(* CODESYS project tesina_IOT.project

Project tree, tasks and I/O mapping:
  Device : CODESYS Control Win V3, 3S - Smart Software Solutions GmbH, version 3.5.12.40
    application Application
      libraries: Standard, * (System); VisuDialogs, * (System)
      task MainTask (cyclic, interval t#20ms, priority 1) calls PLC_PRG
      task VISU_TASK (cyclic, interval 100 ms, priority 31) calls VisuElems.Visu_Prg
      program PLC_PRG [SFC]: Main_active
      function block OOM [ST]
      function block SWITCHER [ST]
      function block ARM_GRID [ST]
      function block ARM_CONTROLLER [ST]
      function block MAIN_CONTROLLER [ST]
      visualisation Visualization
      image pool ImagePool
  text list GlobalTextList
  5ce3da45-db07-42e7-a21c-a00fff4ed8f6|C:\Users\marco\Downloads\Telegram Desktop\abbassato con fusto DX.png
  5ce3da45-db07-42e7-a21c-a00fff4ed8f6|C:\Users\marco\Downloads\Telegram Desktop\abbassato con fusto SX.png
  5ce3da45-db07-42e7-a21c-a00fff4ed8f6|C:\Users\marco\Downloads\Telegram Desktop\alzato con fusto giù DX posizione A.png
  5ce3da45-db07-42e7-a21c-a00fff4ed8f6|C:\Users\marco\Downloads\Telegram Desktop\alzato con fusto giù DX posizione B.png
  5ce3da45-db07-42e7-a21c-a00fff4ed8f6|C:\Users\marco\Downloads\Telegram Desktop\alzato con fusto giù DX posizione C.png
  5ce3da45-db07-42e7-a21c-a00fff4ed8f6|C:\Users\marco\Downloads\Telegram Desktop\alzato con fusto giù SX.png
  5ce3da45-db07-42e7-a21c-a00fff4ed8f6|C:\Users\marco\Downloads\Telegram Desktop\alzato con fusto su DX.png
  5ce3da45-db07-42e7-a21c-a00fff4ed8f6|C:\Users\marco\Downloads\Telegram Desktop\alzato con fusto su SX.png
  5ce3da45-db07-42e7-a21c-a00fff4ed8f6|C:\Users\marco\Downloads\Telegram Desktop\alzato no fusto SX.png
  5ce3da45-db07-42e7-a21c-a00fff4ed8f6|C:\Users\marco\Downloads\Telegram Desktop\alzato posizione 0 - Copia.png
  5ce3da45-db07-42e7-a21c-a00fff4ed8f6|C:\Users\marco\Downloads\Telegram Desktop\alzato con fusto su DX A.png
  5ce3da45-db07-42e7-a21c-a00fff4ed8f6|C:\Users\marco\Downloads\Telegram Desktop\alzato con fusto su DX B.png
  5ce3da45-db07-42e7-a21c-a00fff4ed8f6|C:\Users\marco\Downloads\Telegram Desktop\alzato con fusto su DX C.png
  5ce3da45-db07-42e7-a21c-a00fff4ed8f6|C:\Users\marco\Downloads\Telegram Desktop\alzato con fusto giù DX.png
  5ce3da45-db07-42e7-a21c-a00fff4ed8f6|C:\Users\marco\Desktop\alzato con fusto pos 0.png
*)

// Device/Application/PLC_PRG
PROGRAM PLC_PRG
VAR
	end : OOM();
	grid : ARM_GRID();
	//sensors and stuff
	barcode, geiger : SWITCHER();
	weight: OOM(); //sensor
	start_button: OOM(); //button
	reset_button: OOM(); //button
	light: OOM(); //emergency ligh
	c0 : MAIN_CONTROLLER();
	c1 : ARM_CONTROLLER();
END_VAR

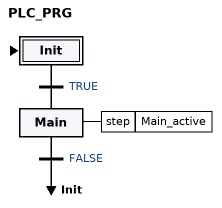
INITIAL_STEP Init:
END_STEP
TRANSITION FROM Init TO Main
    := TRUE;
END_TRANSITION
STEP Main:
    Main_active(N);  // step action
END_STEP
TRANSITION FROM Main TO Init
    := FALSE;
END_TRANSITION

ACTION Main_active:
//INIT
//third level
barcode();
geiger();
weight(); 
start_button();
reset_button();
light();
end();
grid();


c1.grid_input := grid;
c1.hand_input := end;
c1();
end := c1.hand_output;
grid := c1.grid_output;

//first level
c0.arm_controller_input := c1;
c0.barcode_input := barcode;
c0.geiger_input := geiger;
c0.light_input := light;

//solo input per c0
c0.reset_button_input := reset_button;
c0.start_button_input := start_button;
c0.weight_input := weight;

c0();
c1 := c0.arm_controller_output;
barcode := c0.barcode_output;
geiger := c0.geiger_output;
light := c0.light_output;
END_ACTION

END_PROGRAM

// Device/Application/OOM
FUNCTION_BLOCK OOM
// if this class will be used as controller for the  robot hand, we'll assume false as OPEN HAND and true as CLOSED HAND
VAR_INPUT
	stato_in : BOOL := FALSE;
END_VAR
VAR_OUTPUT
	stato_out : BOOL := FALSE;
END_VAR
VAR
	stato : INT := 0;
END_VAR

// 0 idle, 1 off, 2 on
CASE stato OF
	0:
		stato := 1;
		stato_out := FALSE;
		stato_in := FALSE;
	;
	1:
		IF stato_in THEN
			stato := 2;
			stato_out := TRUE;
		END_IF
	;
	2:
		IF NOT stato_in THEN
			stato := 1;
			stato_out := FALSE;
		END_IF
	;
END_CASE

END_FUNCTION_BLOCK

// Device/Application/ARM_GRID
FUNCTION_BLOCK ARM_GRID
VAR_INPUT
	direction : STRING := ''; // 0 or A or B or C or X
END_VAR
VAR_OUTPUT
	current_basket : STRING := '0';
END_VAR
VAR
	status : INT := 1;
	t:TON();
END_VAR

// 0 idle, 1 off, 2 on
CASE status OF
	0: //TR0
		current_basket := 'tr0';
		t(IN := TRUE, PT := T#10S); // emulating transition
		IF  (t.Q = TRUE) THEN // basket 0 reached
			t(IN := FALSE);
			status := 1; //move to starting point on init
		END_IF
	;
	1: // slot 0 starting point
		current_basket := '0';
		IF direction = 'trX' THEN // waiting for new direction's instructions (can be only X from this point)
			status := 5;
		END_IF
	;
	2: // slot A
		t(IN := TRUE, PT := T#10S); // emulating transition
		current_basket := 'trA';
		IF  (t.Q = TRUE) THEN // basket A reached
			t(IN := FALSE);
			status := 7;
		END_IF
	;
	3: // slot B
		t(IN := TRUE, PT := T#10S); // emulating transition
		current_basket := 'trB';
		IF  (t.Q = TRUE) THEN // basket B reached
			t(IN := FALSE);
			status := 8;
		END_IF
	;
	4: // slot C
		t(IN := TRUE, PT := T#10S); // emulating transition
		current_basket := 'trC';
		IF  (t.Q = TRUE) THEN // basket C reached
			t(IN := FALSE);
			status := 9;
		END_IF
	;
	5: // slot X -> grabbing pack
		current_basket := 'trX';
		t(IN := TRUE, PT := T#10S); // emulating transition
		IF  (t.Q = TRUE) THEN // basket X reached
			t(IN := FALSE);
			status := 6;
		END_IF
	;
	6:
		current_basket := 'X';
		// waiting for new direction's instructions (can be everything from this point)
		IF direction = 'trA' THEN
			status := 2;
		ELSIF  direction = 'trB' THEN
			status := 3;
		ELSIF  direction = 'trC' THEN
			status := 4;
		ELSIF  direction = 'tr0' THEN
			status := 0;
		END_IF
	;
	7: //A reached
	current_basket := 'A';
	IF direction = 'tr0' THEN
		status := 0; // to basket number 0
	END_IF
	;
	8: //B reached
	current_basket := 'B';
	IF direction = 'tr0' THEN
		status := 0; // to basket number 0
	END_IF
	;
	9: //C reached
	IF direction = 'tr0' THEN
		status := 0; // to basket number 0
	END_IF
	;
END_CASE

END_FUNCTION_BLOCK

// Device/Application/SWITCHER
FUNCTION_BLOCK SWITCHER
VAR_INPUT
	//active : BOOL := FALSE; //on -> scanning, off -> turned off
	type_simulation : STRING := '';
END_VAR
VAR_OUTPUT
	basket : STRING := 'U'; //values: U (undefined), A, B, C
END_VAR
VAR
	t:TON();
END_VAR

// 0 idle, 1 off, 2 on

IF type_simulation <> 'A' AND type_simulation <> 'B' AND type_simulation <> 'C' THEN
	basket := 'U';
ELSE
	basket := type_simulation;
END_IF

END_FUNCTION_BLOCK

// Device/Application/MAIN_CONTROLLER
FUNCTION_BLOCK MAIN_CONTROLLER
VAR_INPUT
	arm_controller_input : ARM_CONTROLLER();
	barcode_input, geiger_input : SWITCHER();
	weight_input: OOM(); //sensor
	
	start_button_input: OOM(); //button
	reset_button_input: OOM(); //button
	light_input: OOM(); //emergency light
END_VAR
VAR_OUTPUT
	arm_controller_output : ARM_CONTROLLER();
	barcode_output, geiger_output : SWITCHER();

	light_output: OOM(); //emergency light
END_VAR
VAR
	console : STRING := 'init';
	barcode_res, gaiger_res : STRING;
	A_counter, B_counter, C_counter : INT;
	status : INT := 0;
	t:TON();
	//var for UI. true -> invisible
	UI_x, UI_x_grab, UI_x_hold, UI_0, UI_0_W, UI_a_hold, UI_b_hold, UI_c_hold, UI_abc_landed, UI_abc_drop : BOOL := TRUE;
END_VAR

CASE status OF
	0: // INIT
		UI_0 := FALSE;
		IF weight_input.stato_out THEN
			status := 1;
			console := 'sensore di peso attivato, aspettando operatore';
		ELSIF start_button_input.stato_out THEN
			status := 8; //ERROR!
			console := 'bottone premuto ma nulla sul basket. errore!';
		END_IF
		//UI
		IF status <> 0 THEN 
			UI_0 := TRUE;
		END_IF
	;
	1: //s0, weight sensor
		UI_0_W := FALSE;
		IF start_button_input.stato_out THEN
			console := 'bottone premuto, spostamento braccio verso X';
			arm_controller_input.direction := 'trX';
			status := 2;
		END_IF
		//UI
		IF status <> 1 THEN 
			UI_0_W := TRUE;
		END_IF
	;
	2: //TRX
		UI_x := FALSE;
		IF arm_controller_input.position = 'X' THEN
			console := 'braccio ha raggiunto X';
			status := 3;
		END_IF
		//UI
		IF status <> 2 THEN 
			UI_x := TRUE;
		END_IF
	;
	3: //x, timer for grabbing package
		UI_x_grab := FALSE;
		t(IN := TRUE, PT := T#5S);
		console := 'attesa di 5 secondi per la presa del pacco (gestita da c1).';
		IF  (t.Q = TRUE) THEN
			t(IN := FALSE);
			status := 4;
		END_IF
		//UI
		IF status <> 3 THEN
			UI_x_grab := TRUE;	
		END_IF
	;
	4: //scan
		UI_x_hold := FALSE;
		IF barcode_input.basket = 'A' OR barcode_input.basket = 'B' OR barcode_input.basket = 'C' THEN
			console := 'scansione barcode pacco completata correttamente';
			status := 5;
			barcode_res := barcode_input.basket;
		ELSIF barcode_input.basket = 'U' THEN
			console := 'scansione barcode fallita, pacco uknown';
			status := 9;
		END_IF
		//UI
		IF status <> 4 THEN
			UI_x_hold := TRUE;			
		END_IF
	;
	5: //verify
		UI_x_hold := FALSE;
		gaiger_res := geiger_output.basket;
		IF gaiger_res = 'U' OR gaiger_res <> barcode_res THEN
			console := 'scansione radioattività fallita, unknown o diverso dal barcode';
			status := 9;
		ELSIF gaiger_res = 'A' THEN //package A
			console := 'scansioni completate: analisi pacco A';
			IF A_counter > 4 THEN
				status := 9; // full
				console := 'nastro trasportatore A pieno. errore';
			ELSE
				A_counter := A_counter + 1;
				arm_controller_input.direction := 'trA';
				console := 'avviato braccio verso nastro A, incrementato contatore';
				status := 10; 
			END_IF
		ELSIF gaiger_res = 'B' THEN //package B
			console := 'scansioni completate: analisi pacco B';
			IF B_counter > 4 THEN
				console := 'nastro trasportatore B pieno. errore';
				status := 9; // full
			ELSE
				B_counter := B_counter + 1;
				arm_controller_input.direction := 'trB';
				status := 11; 
				console := 'avviato braccio verso nastro B, incrementato contatore';
			END_IF
		ELSIF gaiger_res = 'C' THEN //package C
			console := 'scansioni completate: analisi pacco C';
			IF C_counter > 4 THEN
				status := 9; // full
				console := 'nastro trasportatore C pieno. errore';
			ELSE
				C_counter := C_counter + 1;
				arm_controller_input.direction := 'trC';
				status := 12; 
				console := 'avviato pacco verso nastro C, incrementato contatore';
			END_IF
		END_IF
		//UI
		IF status <> 5 THEN
			UI_x_hold := TRUE;			
		END_IF
	;
	6:
		UI_abc_landed := FALSE;
		console := 'attesa 5 secondi sgancio pacco in postazione';
		t(IN := TRUE, PT := T#5S);
		IF  (t.Q = TRUE) THEN
			t(IN := FALSE);
			status := 7;
		END_IF
		//UI
		IF status <> 6 THEN 
			UI_abc_landed := TRUE;
		END_IF
	;
	7:
		UI_abc_drop := FALSE;
		console := 'sgancio completato, redirezionamento braccio verso tr0';
		arm_controller_input.direction := 'tr0';
		status := 13;
		//UI
		IF status <> 7 THEN 
			UI_abc_drop := TRUE;
		END_IF
	;
	
	/////////////////
	// ERROR SECTION
	////////////////
	8: //B0 ERR, start_button pushed before weight sensor is ok
		UI_0 := FALSE;
		light_input.stato_in := TRUE;
		IF reset_button_input.stato_out THEN
			light_input.stato_in := FALSE;
			console := 'bottone di reset premuto, siamo tornati ad init';
			status := 0;
		END_IF
		//UI
		IF status <> 8 THEN 
			UI_0 := TRUE;
		END_IF
	;
	9: //ERROR come case 8 ma riporto il braccio in posizione 0 e quando resetto assumo di aver svuotato i rulli
		UI_0 := FALSE;
		light_input.stato_in := TRUE;
		arm_controller_input.direction := 'tr0'; //questo dovrebbe essere colto come errore da arm controller, passaggio da X -> tr0
		IF reset_button_input.stato_out AND arm_controller_input.position = '0' THEN
			light_input.stato_in := FALSE;
			A_counter := 0;
			B_counter := 0;
			C_counter := 0;
			console := 'braccio è in 0, slot svuotati, bottone di reset premuto, siamo tornati ad init';
			status := 0;
		END_IF
		//UI
		IF status <> 9 THEN 
			UI_0 := TRUE;
		END_IF
	;
	//////////////
	// END ERRORS
	/////////////
	
	10:
		UI_a_hold := FALSE;
		IF arm_controller_input.position = 'A' THEN
			console := 'postazione A raggiunta';
			status := 6;
		END_IF
		//UI
		IF status <> 10 THEN
			UI_a_hold := TRUE;			
		END_IF
	;
	11:
		UI_b_hold := FALSE;
		IF arm_controller_input.position = 'B' THEN
			console := 'postazione B raggiunta';
			status := 6;
		END_IF
		//UI
		IF status <> 11 THEN
			UI_b_hold := TRUE;			
		END_IF
	;
	12:
		UI_c_hold := FALSE;
		IF arm_controller_input.position = 'C' THEN
			console := 'postazione C raggiunta';
			status := 6;
		END_IF
		//UI
		IF status <> 12 THEN
			UI_c_hold := TRUE;			
		END_IF
	;
	13:
		UI_0 := FALSE;
		IF arm_controller_input.position = '0' THEN
			console := 'postazione 0 raggiunta. siamo tornati ad init';
			status := 0;
		END_IF
		//UI
		IF status <> 13 THEN
			UI_0 := TRUE;			
		END_IF
	;
END_CASE

//updating values
arm_controller_output := arm_controller_input;
barcode_output := barcode_input;
geiger_output := geiger_input;
light_output := light_input;

END_FUNCTION_BLOCK

// Device/Application/ARM_CONTROLLER
FUNCTION_BLOCK ARM_CONTROLLER
VAR_INPUT
	direction : STRING := 'INIT';
	grid_input : ARM_GRID();
	hand_input : OOM();
	//c0_input : MAIN_CONTROLLER();
END_VAR
VAR_OUTPUT
	position : STRING := '';
	grid_output : ARM_GRID();
	hand_output : OOM();
	//c0_output : MAIN_CONTROLLER();
END_VAR
VAR
	status : INT := 0;
END_VAR

CASE status OF
	0:	//INIT
		IF direction = 'trX' THEN //moving grid to trX and 
			grid_input.direction := 'trX';
			status := 1;
		END_IF
	;
	1: //TRX
		IF grid_input.current_basket = 'X' THEN
			hand_input.stato_in := TRUE;
			position := 'X';
			status := 2;
		END_IF
	;
	2: //X
		IF direction = 'trA' THEN //moving grid to trA 
			grid_input.direction := 'trA';
			status := 3; //A
		ELSIF direction = 'trB' THEN //moving grid to trB  
			grid_input.direction := 'trB';
			status := 4; //B
		ELSIF direction = 'trC' THEN //moving grid to trC  
			grid_input.direction := 'trC';
			status := 5; //C
		ELSIF direction = 'tr0' THEN //ERROR DETECTED!! 
			//it's like case 6
			grid_input.direction := 'tr0';
			status := 7; // waiting for destination reached
		END_IF
	;
	3: //A
		IF grid_input.current_basket = 'A' THEN
			hand_input.stato_in := FALSE; 
			position := 'A';
			status := 6; //GOING TO WAIT RESET
		END_IF
	;
	4: //B
		IF grid_input.current_basket = 'B' THEN
			hand_input.stato_in := FALSE; 
			position := 'B';
			status := 6; //GOING TO WAIT RESET
		END_IF		
	;
	5: //C
		IF grid_input.current_basket = 'C' THEN
			hand_input.stato_in := FALSE; 
			position := 'C';
			status := 6; //GOING TO WAIT RESET
		END_IF
	;
	6: //WAITING FOR RESET
		IF direction = 'tr0' THEN //moving grid to tr0 
			grid_input.direction := 'tr0';
			status := 7; //WAITING FOR TR0
		END_IF
	;
	7: // WHEN 0 IS REACHED WE SWITCH TO INIT
		IF grid_input.current_basket = '0' THEN
			position := '0';
			status := 0; // init
		END_IF
	;	
END_CASE

grid_output := grid_input;
hand_output := hand_input;

END_FUNCTION_BLOCK

// Device/Application/Visualization
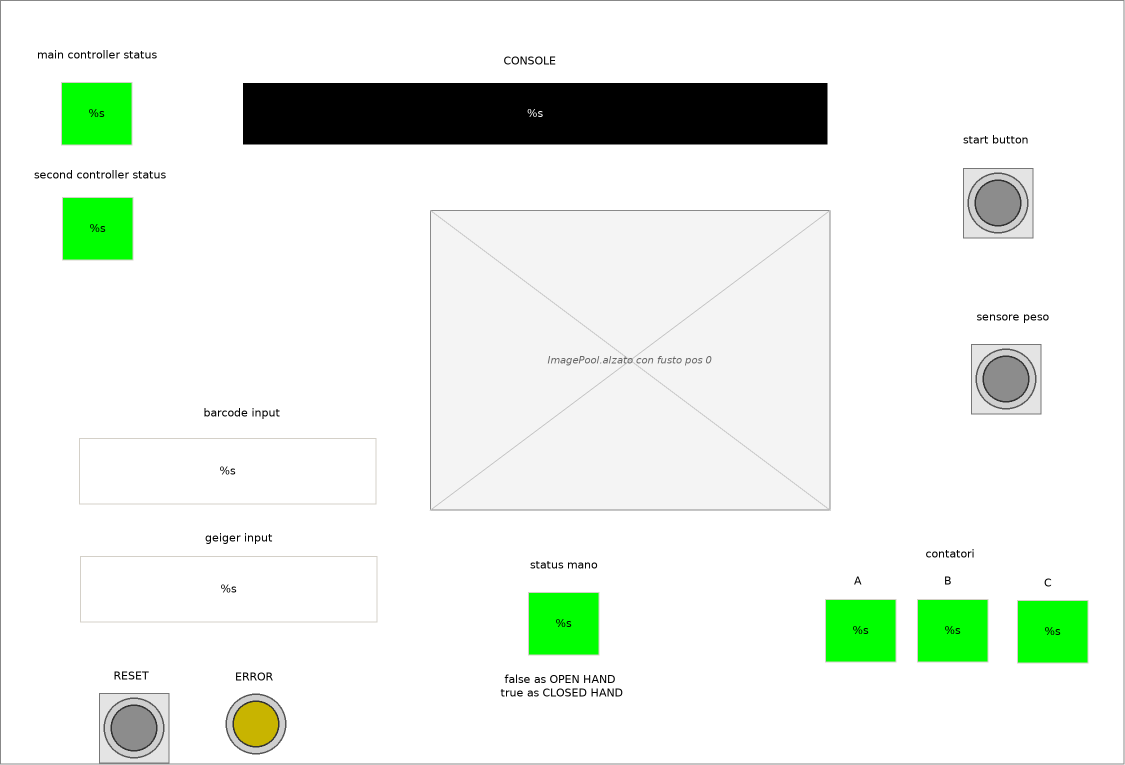
VISUALIZATION Visualization  // 1125x765
    Textfield (61,82 71x63), "%s", text variable: PLC_PRG.c0.status
    Textfield (79,438 297x66), "%s", text variable: PLC_PRG.barcode.type_simulation
        OnMouseClick: write the text variable via Default
    Textfield (80,556 297x66), "%s", text variable: PLC_PRG.geiger.type_simulation
        OnMouseClick: write the text variable via Default
    Label (167,398 150x30), "barcode input"
    Label (164,523 150x30), "geiger input"
    Label (22,40 150x30), "main controller status"
    PushSwitchLed (963,168 70x70), variable: PLC_PRG.start_button.stato_in, behaviour: TOGGLE, style: Switch-PushSwitchLed-Gray
    Label (921,125 150x30), "start button"
    Label (938,302 150x30), "sensore peso"
    PushSwitchLed (971,344 70x70), variable: PLC_PRG.weight.stato_in, behaviour: TOGGLE, style: Switch-PushSwitchLed-Gray
    Textfield (62,197 71x63), "%s", text variable: PLC_PRG.c1.status
    Label (25,160 150x30), "second controller status"
    Textfield (242,82 586x63), "%s", text variable: PLC_PRG.c0.console
    Label (455,46 150x30), "CONSOLE"
    Textfield (528,592 71x63), "%s", text variable: PLC_PRG.end.stato_out
    Label (489,550 150x30), "status mano"
    Textfield (825,599 71x63), "%s", text variable: PLC_PRG.c0.A_counter
    Label (783,566 150x30), "A"
    PushSwitchLed (99,693 70x70), variable: PLC_PRG.reset_button.stato_in, behaviour: TOGGLE, style: Switch-PushSwitchLed-Gray
    Label (56,661 150x30), "RESET"
    Lamp1 (221,689 70x70), variable: PLC_PRG.light.stato_out, style: Lamp-Lamp1-Yellow
    Label (179,662 150x30), "ERROR"
    Label (489,658 146x56), "false as OPEN HAND true as CLOSED HAND"
    Textfield (917,599 71x63), "%s", text variable: PLC_PRG.c0.B_counter
    Label (873,566 150x30), "B"
    Textfield (1017,600 71x63), "%s", text variable: PLC_PRG.c0.C_counter
    Label (973,568 150x30), "C"
    Label (875,539 150x30), "contatori"
    Image (430,210 400x300), invisible if: PLC_PRG.c0.UI_0, image: ImagePool.alzato posizione 0 - Copia
    Image (430,210 400x300), invisible if: PLC_PRG.c0.UI_x, image: ImagePool.alzato con fusto giù SX
    Image (430,210 400x300), invisible if: PLC_PRG.c0.UI_x_grab, image: ImagePool.abbassato con fusto SX
    Image (430,210 400x300), invisible if: PLC_PRG.c0.UI_x_hold, image: ImagePool.alzato con fusto su SX
    Image (430,210 400x300), invisible if: PLC_PRG.c0.UI_a_hold, image: ImagePool.alzato con fusto su DX A
    Image (430,210 400x300), invisible if: PLC_PRG.c0.UI_b_hold, image: ImagePool.alzato con fusto su DX B
    Image (430,210 400x300), invisible if: PLC_PRG.c0.UI_c_hold, image: ImagePool.alzato con fusto su DX C
    Image (430,210 400x300), invisible if: PLC_PRG.c0.UI_abc_drop, image: ImagePool.alzato con fusto giù DX
    Image (430,210 400x300), invisible if: PLC_PRG.c0.UI_abc_landed, image: ImagePool.abbassato con fusto DX
    Image (430,210 400x300), invisible if: PLC_PRG.c0.UI_0_W, image: ImagePool.alzato con fusto pos 0
END_VISUALIZATION
